// Mitsubishi GX Works2 project: contador com switch aberto   PLC: Q03UDV

PROGRAM MAIN
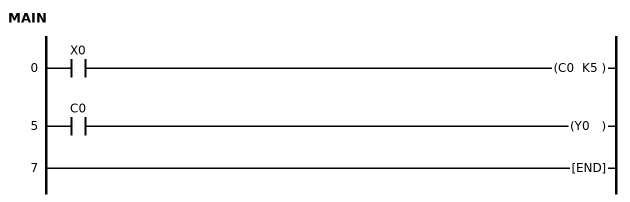
0     LD      X0
      OUT     C0 K5
5     LD      C0
      OUT     Y0
7     END
END_PROGRAM
